// TIA Portal V16 export
// export: Created 2021-09-08T12:44:31.3105867Z, ExportSetting WithDefaults, DisplayName Totally Integrated Automation Portal, DisplayVersion V16 Update 3, DisplayName TIA Portal Version Control Interface, DisplayVersion V16 Update 2, DisplayName TIA Portal Openness, DisplayVersion V16 Update 3, DisplayName TIA Portal Teamcenter Gateway, DisplayVersion V16, DisplayName STEP 7 Professional, DisplayVersion V16 Update 3, DisplayName STEP 7 Safety, DisplayVersion V16, DisplayName WinCC Advanced, DisplayVersion V16 Update 3
VAR_GLOBAL   // PLC tag table "Default tag table"
   System_Byte AT %MB1 : Byte;
   FirstScan AT %M1.0 : Bool;
   DiagStatusUpdate AT %M1.1 : Bool;
   AlwaysTRUE AT %M1.2 : Bool;
   AlwaysFALSE AT %M1.3 : Bool;
   Clock_Byte AT %MB0 : Byte;
   Clock_10Hz AT %M0.0 : Bool;
   Clock_5Hz AT %M0.1 : Bool;
   "Clock_2.5Hz" AT %M0.2 : Bool;
   Clock_2Hz AT %M0.3 : Bool;
   "Clock_1.25Hz" AT %M0.4 : Bool;
   Clock_1Hz AT %M0.5 : Bool;
   "Clock_0.625Hz" AT %M0.6 : Bool;
   "Clock_0.5Hz" AT %M0.7 : Bool;
   ClockOneSycle AT %MB2 : Byte;
   ClockOneCycle10HZ AT %M2.0 : Bool;
   ClockOneCycle5HZ AT %M2.1 : Bool;
   ClockOneCycle2_5HZ AT %M2.2 : Bool;
   ClockOneCycle2HZ AT %M2.3 : Bool;
   ClockOneCycle1_25HZ AT %M2.4 : Bool;
   ClockOneCycle1HZ AT %M2.5 : Bool;
   ClockOneCycle0_65HZ AT %M2.6 : Bool;
   ClockOneCycle0_5HZ AT %M2.7 : Bool;
END_VAR
